INTERFACE I_Counter

METHOD Increment : BOOL
END_METHOD

PROPERTY Step : DINT
GET
END_GET
SET
END_SET
END_PROPERTY

END_INTERFACE

(* stored: Version 1.1.0.1, ProductVersion 3.1.4024.12
   Itf I_Counter: Id {5f1c2d9e-0a6b-4c11-9d3e-7a1b2c3d4e10}
   Method Increment: Id {5f1c2d9e-0a6b-4c11-9d3e-7a1b2c3d4e11}
   Property Step: Id {5f1c2d9e-0a6b-4c11-9d3e-7a1b2c3d4e12}
   Get Get: Id {5f1c2d9e-0a6b-4c11-9d3e-7a1b2c3d4e13}
   Set Set: Id {5f1c2d9e-0a6b-4c11-9d3e-7a1b2c3d4e14} *)
